FUNCTION F_IsError : BOOL
VAR_INPUT
    fb : FB_Motor;
END_VAR

F_IsError := fb.nErrorId <> 0;

END_FUNCTION

(* stored: Version 1.1.0.1, ProductVersion 3.1.4024.12
   POU F_IsError: Id {a1b2c3d4-0011-4000-8000-000000000011}, SpecialFunc None *)
